PROGRAM TCP_IP
VAR
END_VAR

END_PROGRAM

(* stored: Version 1.1.0.1, ProductVersion 3.1.4024.0
   POU TCP_IP: Id {b3a78b8f-7402-46f3-942d-2e14f4eca26b}, SpecialFunc None *)
